// TwinCAT 3 PLC project Listener
// ProgramVersion: 3.1.4021.2
// libraries:
//   Tc2_Standard, * (Beckhoff Automation GmbH)
//   Tc2_System, * (Beckhoff Automation GmbH)
//   Tc3_EventLogger, * (Beckhoff Automation GmbH)
//   Tc3_Module, * (Beckhoff Automation GmbH)
// project tree:
//   / ListenerTask.TcTTO (not stored)
//   POUs/ FB_ListenerTest.TcPOU, MAIN.TcPOU, FB_SampleListener.TcPOU
// (motion and I/O tree: see PLC project publisher)
// real-time tasks:
//   TASK PublisherTask: cycle T#10ms, priority 20, ADS port 350
//   TASK ListenerTask: cycle T#10ms, priority 1, ADS port 351

// ---- POUs/FB_ListenerTest.TcPOU
FUNCTION_BLOCK FB_ListenerTest
VAR_INPUT
END_VAR
VAR_OUTPUT
END_VAR
VAR
	hr : HRESULT;
	
	bSubscribe : BOOL := TRUE;
	bSubscribed : BOOL;
	bUnSubscribe : BOOL;
	
	fbListenerFilter : FB_TcEventFilter; 
	fbMessageListener : FB_SampleListener;
END_VAR

fbMessageListener.Execute(); // retrieve messages and its texts


IF bSubscribe THEN 
	bSubscribe := FALSE;
	fbListenerFilter.Clear().EventClass.EqualTo(TC_EVENTS.PublisherEventClass.Message.uuidEventClass); //define all events (messages and alarms) from this eventclass   
	hr := fbMessageListener.Subscribe2(fbListenerFilter); //subscribe to retrieve defined events
	bSubscribed := fbMessageListener.bSubscribed;

END_IF 

IF bUnSubscribe THEN 
	bUnSubscribe := FALSE;
	hr := fbMessageListener.Unsubscribe();
	bSubscribed := fbMessageListener.bSubscribed;

END_IF

END_FUNCTION_BLOCK

// ---- POUs/FB_SampleListener.TcPOU
FUNCTION_BLOCK FB_SampleListener EXTENDS FB_ListenerBase2
VAR_INPUT
END_VAR
VAR_OUTPUT
END_VAR
VAR
	sJsonAttribute : STRING (10000);	
	hr : HRESULT;
	
	nCntMessagesSent : INT;
	nCntAlarmsRaised : INT;
	nCntAlarmsConfirmed : INT;
	nCntAlarmsCleared : INT;
	
	//text retrieval of message
	fbRequestEventText : FB_RequestEventText;
	{attribute 'TcEncoding':='UTF-8'}
	sLastMessageText : STRING;
	bReqText : BOOL;
END_VAR

METHOD Execute : HRESULT
VAR_INPUT
END_VAR
Execute := SUPER^.Execute(); //retrieve events

//retrieve the text of a message
IF 	bReqText AND fbRequestEventText.bError THEN 
	sLastMessageText := 'Error';
	bReqText := FALSE; 
ELSIF bReqText AND NOT  fbRequestEventText.bBusy THEN
	fbRequestEventText.GetString(sLastMessageText, SIZEOF(sLastMessageText));
	bReqText := FALSE;
END_IF
END_METHOD

METHOD OnAlarmCleared : HRESULT
VAR_INPUT
	fbEvent : REFERENCE TO FB_TcEvent;
END_VAR
nCntAlarmsCleared := nCntAlarmsCleared + 1;

OnAlarmCleared := S_OK; // in order to receive more callbacks (Set <> S_OK in order to cancel the callbacks for this program cycle.)
END_METHOD

METHOD OnAlarmConfirmed : HRESULT
VAR_INPUT
	fbEvent : REFERENCE TO FB_TcEvent;
END_VAR
nCntAlarmsConfirmed := nCntAlarmsConfirmed + 1;

OnAlarmConfirmed := S_OK; // in order to receive more callbacks (Set <> S_OK in order to cancel the callbacks for this program cycle.)
END_METHOD

METHOD OnAlarmRaised : HRESULT
VAR_INPUT
	fbEvent : REFERENCE TO FB_TcEvent;
END_VAR
hr := fbEvent.GetJsonAttribute(sJsonAttribute, SIZEOF(sJsonAttribute));
nCntAlarmsRaised := nCntAlarmsRaised + 1;

OnAlarmRaised := S_OK; // in order to receive more callbacks (Set <> S_OK in order to cancel the callbacks for this program cycle.)
END_METHOD

METHOD OnMessageSent : HRESULT
VAR_INPUT
	fbEvent : REFERENCE TO FB_TcEvent;
END_VAR

VAR 
END_VAR
hr := fbEvent.GetJsonAttribute(sJsonAttribute, SIZEOF(sJsonAttribute));
nCntMessagesSent := nCntMessagesSent + 1;

fbRequestEventText.Request(eventClass:=fbEvent.EventClass, nEventId:=fbEvent.nEventId, nLangId:=TcLcid.en_US, ipArgs:=fbEvent.ipArguments );
bReqText := TRUE;

OnMessageSent := S_OK; // in order to receive more callbacks (Set <> S_OK in order to cancel the callbacks for this program cycle.)
END_METHOD

END_FUNCTION_BLOCK

// ---- POUs/MAIN.TcPOU
PROGRAM MAIN
VAR
	fbListenerTest : FB_ListenerTest;
END_VAR

fbListenerTest();

END_PROGRAM
